// Brief: Master Arm MasterSlave controller
FUNCTION_BLOCK PUBLIC FB_StateCtrlMasterSlave EXTENDS FB_MasterArmCtrlBase
VAR_INPUT
END_VAR
VAR_OUTPUT
END_VAR
VAR
	// joint4 controller
	m_redunJntCtrl : FB_RedunJntControl;
	
	// flag if project joint4 torque to nullspace
	m_nullspaceCtrl : BOOL :=FALSE;
	
	// boundary limit force feedback
	m_boundaryForce : FB_boundaryForceFeedback;
	
	// joint torque for master-slave error
	m_boundaryTrq :Vec7d;
	
	// friction compensation scale
	m_frictionCompScale :LREAL :=1.0;

END_VAR

// override this function in each exact controller
METHOD PROTECTED calcCmdJntPos : BOOL

VAR_IN_OUT CONSTANT
	i_slaveIdx :INT;
	i_shoulderPose :ST_Frame;
	i_masterArm :FB_MasterArm;
	i_slaveStatus :ST_SlaveStatus;
END_VAR
VAR 

END_VAR
IF i_slaveStatus.m_instruStauts[i_slaveIdx].m_type = InstruType_UltrasoundKnifeS OR 
	i_slaveStatus.m_instruStauts[i_slaveIdx].m_type = InstruType_UltrasoundKnifeU THEN
	calcCmdJntPos_USKnife(i_slaveIdx,i_shoulderPose,i_masterArm,i_slaveStatus);
ELSE
	calcCmdJntPos_BasicInstru(i_slaveIdx,i_shoulderPose,i_masterArm,i_slaveStatus);
END_IF
END_METHOD

// override this function in each exact controller
METHOD PROTECTED calcCmdJntPos_BasicInstru : BOOL

VAR_IN_OUT CONSTANT
	i_slaveIdx :INT;
	i_shoulderPose :ST_Frame;
	i_masterArm :FB_MasterArm;
	i_slaveStatus :ST_SlaveStatus;
END_VAR
VAR 

END_VAR
m_cmdJntPos:=i_masterArm.curJntPos;
m_cmdJntVel:=i_masterArm.curJntVel;
m_cmdCartPose:=i_masterArm.curCartPose;
END_METHOD

// override this function in each exact controller
METHOD PROTECTED calcCmdJntPos_USKnife : BOOL

VAR_IN_OUT CONSTANT
	i_slaveIdx :INT;
	i_shoulderPose :ST_Frame;
	i_masterArm :FB_MasterArm;
	i_slaveStatus :ST_SlaveStatus;
END_VAR
VAR CONSTANT
	// orientation tracking parameters
	m_rotTrackKp : LREAL := 200;
	m_maxTrackVel :LREAL := PI;
	m_trackAngThres :LREAL := 2* g_deg2rad;
END_VAR
VAR 
	cartTrackVel :Vec3d;
	i,j : INT;
	invRot :Mat3d;
	cmdRotInView:Mat3d;
	rotT,rotErr :Mat3d;
	angle:LREAL;
	axis:Vec3d;
	
	oriJaco:Mat34;
	oriJt:Mat43;
	oriJJt:Mat3d;
	oriJJtInv:Mat3d;
	oriJPinv:Mat43;
	jntTrackVel:Vec4d;
	JpinvJ, nullJ:Mat4d;
	eye4d :Mat4d := g_eye4d;
	redunCtrlVel :Vec4d;
	jnt4TrackVel :LREAL;
	cmdZAxis, curZAxis :Vec3d;
END_VAR
m_jntOPMode[1] := DriverOPMode_Trq;
m_jntOPMode[2] := DriverOPMode_Trq;
m_jntOPMode[3] := DriverOPMode_Trq;
m_jntOPMode[4] := DriverOPMode_PosTrq;
m_jntOPMode[5] := DriverOPMode_PosTrq;
m_jntOPMode[6] := DriverOPMode_PosTrq;
m_jntOPMode[7] := DriverOPMode_Trq;

// use matched slave arm orientation as target, 
//	and transform from view coordinate to arm coordinate 
cmdRotInView := i_slaveStatus.m_curArmPose[i_slaveIdx].m_rot;
matTranspose(i_shoulderPose.m_rot, invRot);
matMultiply(invRot, cmdRotInView, m_cmdCartPose.m_rot);
m_cmdCartPose.m_pos:= i_masterArm.curCartPose.m_pos;

// first three joints and joint7 is passive control
FOR i:=1 TO 3 DO 
	m_cmdJntPos[i]:=i_masterArm.curJntPos[i];
	m_cmdJntVel[i]:=i_masterArm.curJntVel[i];
END_FOR
m_cmdJntPos[7]:=i_masterArm.curJntPos[7];
m_cmdJntVel[7]:=i_masterArm.curJntVel[7];

// compute cartesian tracking velocity
FOR i:=1 TO 3 DO
	cmdZAxis[i] :=  m_cmdCartPose.m_rot[i,3];
	curZAxis[i] := i_masterArm.simCartPose.m_rot[i,3];
END_FOR
angle := ACOS(LIMIT(-1,vecDot(cmdZAxis,curZAxis),1));
axis := cross(curZAxis, cmdZAxis);
IF ABS(angle)> g_smallAng AND ABS(angle-pi)> g_smallAng THEN
	normalize(axis);
END_IF
vecMultiNum(axis, LIMIT(-m_maxTrackVel, angle*m_rotTrackKp, m_maxTrackVel), cartTrackVel);

// compute pinv of orientation jacobian
FOR i:=1 TO 3 DO
	FOR j:=1 TO 4 DO
		oriJaco[i,j]:=i_masterArm.simJaco[i+3,j+3];
	END_FOR
END_FOR
matTranspose(oriJaco, oriJt);
matMultiply(oriJaco ,oriJt , oriJJt);
invMat3(oriJJt, oriJJtInv);
matMultiply(oriJt, oriJJtInv, oriJPinv);
matMultiVec(oriJpinv, cartTrackVel, jntTrackVel);

// calculate nullspace
matMultiply(oriJPinv, oriJaco, JpinvJ);
matSub(eye4d , JpinvJ, nullJ);

// redundant velocity
jnt4TrackVel:=calcRedunVel(i_masterArm);
redunCtrlVel[1]:=nullJ[1,1]*jnt4TrackVel;
redunCtrlVel[2]:=nullJ[2,1]*jnt4TrackVel;
redunCtrlVel[3]:=nullJ[3,1]*jnt4TrackVel;
redunCtrlVel[4]:=nullJ[4,1]*jnt4TrackVel;

// update final command joint position and velocity
FOR i :=1 TO 3 DO 
	m_cmdJntVel[i+3]:=jntTrackVel[i]+redunCtrlVel[i];
	m_cmdJntPos[i+3]:=m_cmdJntPos[i+3]+m_cmdJntVel[i+3]*g_armCtrlCycleTime;
END_FOR
END_METHOD

// override this function in each exact controller
METHOD PROTECTED calcCmdJntTrq : BOOL

VAR_IN_OUT CONSTANT
	i_slaveIdx :INT;
	i_shoulderPose :ST_Frame;
	i_masterArm :FB_MasterArm;
	i_slaveStatus :ST_SlaveStatus;
END_VAR

VAR 
	
END_VAR
IF i_slaveStatus.m_instruStauts[i_slaveIdx].m_type = InstruType_UltrasoundKnifeS OR 
	i_slaveStatus.m_instruStauts[i_slaveIdx].m_type = InstruType_UltrasoundKnifeU THEN
	calcCmdJntTrq_USKnife(i_slaveIdx,i_shoulderPose,i_masterArm,i_slaveStatus);
ELSE
	calcCmdJntTrq_BasicInstru(i_slaveIdx,i_shoulderPose,i_masterArm,i_slaveStatus);
END_IF
END_METHOD

// override this function in each exact controller
METHOD PROTECTED calcCmdJntTrq_BasicInstru : BOOL

VAR_IN_OUT CONSTANT
	i_slaveIdx :INT;
	i_shoulderPose :ST_Frame;
	i_masterArm :FB_MasterArm;
	i_slaveStatus :ST_SlaveStatus;
END_VAR

VAR 
	nullspaceMat :Mat7d;
	ctrlTrq : Vec7d;
	boundaryTrq :Vec7d;
	withinBoundary :BOOL;
	i :INT;
	inertiaTrq:LREAL;
END_VAR
// boundary force feedback
m_boundaryTrq :=m_boundaryForce.run(i_slaveIdx, i_shoulderPose, i_masterArm, i_slaveStatus);
withinBoundary := (norm(m_boundaryTrq)<g_smallNum);

// redundant joint4 controller
ctrlTrq := g_zeroVec7d;
ctrlTrq[4] := m_redunJntCtrl.run(i_masterArm, i_followEnable:=withinBoundary);

// project to nullspace
IF m_nullspaceCtrl THEN
	nullspaceMat:=i_masterArm.dynaNullspace;
	matMultiVec(nullspaceMat,ctrlTrq, m_cmdJntTrq);
	vecSelfMultiNum(m_cmdJntTrq, ctrlTrq[4] / m_cmdJntTrq[4]);
ELSE
	m_cmdJntTrq := ctrlTrq;
END_IF

// add friction compensation
FOR i:=1 TO g_mJntNum DO 
	m_cmdJntTrq[i] := m_cmdJntTrq[i] +m_frictionCompScale * i_masterArm.jntFriction[i] + m_boundaryTrq[i]+i_masterArm.jntExtTrq[i];
END_FOR
END_METHOD

// override this function in each exact controller
METHOD PROTECTED calcCmdJntTrq_USKnife : BOOL

VAR_IN_OUT CONSTANT
	i_slaveIdx :INT;
	i_shoulderPose :ST_Frame;
	i_masterArm :FB_MasterArm;
	i_slaveStatus :ST_SlaveStatus;
END_VAR

VAR 
	i :INT;
END_VAR
m_cmdJntTrq :=g_zeroVec7d;
// boundary force feedback
m_boundaryTrq :=m_boundaryForce.run(i_slaveIdx, i_shoulderPose, i_masterArm, i_slaveStatus);
m_cmdJntTrq[7] := m_boundaryTrq[7];
END_METHOD

METHOD PROTECTED calcRedunVel : LREAL
VAR_IN_OUT CONSTANT
	i_masterArm :FB_MasterArm;
END_VAR

VAR 
	// redundant control parameters
	m_jnt4AdjustKp : LREAL :=10;
	m_jnt4MaxVel :LREAL :=pi/3 ;
	m_linearVelLb :LREAL := 0.02;
	m_linearVelUb :LREAL :=0.1;	
	
	j6Bias,j5Bias :LREAL;
	velScale :LREAL;
	linearVel :Vec3d;
	curJntPos : Vec7d;
	jnt4LinkPos :LREAL;
END_VAR
// compute desired joint4 link position
curJntPos :=  i_masterArm.cmdJntPos;
jnt4LinkPos:=i_masterArm.jnt4MotorToLink(curJntPos[2],curJntPos[3],curJntPos[4]);
IF 1= i_masterArm.armIdx THEN
	j6Bias :=curJntPos[6]+PI/2;
ELSE 
	j6Bias := curJntPos[6]-PI/2;
END_IF

// scale based on joint5 position
j5Bias :=  LIMIT (0, ABS(curJntPos[5] -pi), pi/2);
j6Bias := j6Bias * ABS(COS(j5Bias));

// scale based on linear velocity
linearVel[1]:=i_masterArm.curCartTwist[1];
linearVel[2]:=i_masterArm.curCartTwist[2];
linearVel[3]:=i_masterArm.curCartTwist[3];
velScale :=LIMIT(0, (norm(linearVel)-m_linearVelLb)/(m_linearVelUb-m_linearVelLb),1.0);


calcRedunVel := LIMIT(-m_jnt4MaxVel, -j6Bias * m_jnt4AdjustKp * velScale ,m_jnt4MaxVel);

// joint limit
IF (calcRedunVel > 0 AND jnt4LinkPos+calcRedunVel * g_armCtrlCycleTime > GVL_ArmJointParameters.g_maxJntPos[i_masterArm.armIdx,4])
	 OR ( calcRedunVel <0 AND  jnt4LinkPos +calcRedunVel * g_armCtrlCycleTime< GVL_ArmJointParameters.g_minJntPos[i_masterArm.armIdx,4]) THEN
	 calcRedunVel :=0;
END_IF
END_METHOD

METHOD PUBLIC init : BOOL
VAR_IN_OUT CONSTANT
	i_masterArm	:FB_MasterArm;
END_VAR
VAR_IN_OUT 
	r_masterArmCtrlCmd :ST_ArmCtrlCmds;
END_VAR

VAR
	i:INT;
END_VAR
SUPER^.Init(i_masterArm,r_masterArmCtrlCmd);

m_jntOPMode := g_allTrqMode;
//m_jntOPMode := g_allPosMode;

// init controller
m_redunJntCtrl.init(i_masterArm);

// update commands to arm
copyCmds(r_masterArmCtrlCmd);
END_METHOD

END_FUNCTION_BLOCK

(* stored: Version 1.1.0.1, ProductVersion 3.1.4024.11
   POU FB_StateCtrlMasterSlave: Id {5b96f309-da76-444d-a9fb-2d4321895cd7}, SpecialFunc None
   Method calcCmdJntPos: Id {b549ed00-ec1a-412a-94d0-63a741bf9608}
   Method calcCmdJntPos_BasicInstru: Id {239c44da-fbb4-4bf5-8dd0-8022d66af60b}
   Method calcCmdJntPos_USKnife: Id {e3490571-181c-4e3a-9266-10457d84eb98}
   Method calcCmdJntTrq: Id {590b7c96-65ed-47d5-8eb2-8a13ee8a5533}
   Method calcCmdJntTrq_BasicInstru: Id {924c67b8-8dc8-4b14-a8ff-535af80c10ba}
   Method calcCmdJntTrq_USKnife: Id {89963b71-7e72-4bb1-9f43-b099432ea948}
   Method calcRedunVel: Id {2d8bb2ec-2a44-4bc5-9d2d-80c4739e4cf3}
   Method init: Id {1bea1de4-0538-46fc-be44-e671d6da03c3} *)
